INTERFACE I_EnumDatatypeAddedEvent EXTENDS I_Event

PROPERTY PUBLIC Target : I_EnumDatatype
GET
END_GET
END_PROPERTY

END_INTERFACE

(* stored: Version 1.1.0.1, ProductVersion 3.1.4024.12
   Itf I_EnumDatatypeAddedEvent: Id {b2d93485-faac-01a2-17ae-eccaec3c33aa}
   Property Target: Id {6a189a51-53ae-0ce9-3244-1f0780293b6a}
   Get Get: Id {dc08815f-0da6-0ce0-0a9a-04bce20feb3d} *)
